Omron CX-Programmer project NewProject (CX-Programmer 9.73)

# PLC FINAL: CS1G CPU42

## Global symbols (name address type ; comment)
C0001 BOOL  ; Reset
C0005 BOOL  ; Brojac ponavljaja
T0001 BOOL  ; Zeleno iskljuceno pesacima
T0002 BOOL  ; Crveno iskljuceno pesacima
T0003 BOOL  ; Zuto iskljuceno kolima
T0004 BOOL  ; Zeleno iskljuceno kolima
T0005 BOOL  ; Brojac

## Program NewProgram1 (cyclic task 0)
Local symbols
Crveno_Pesaci 2961.02 BOOL  ; Pesaci crveno
Crveno_Voz 2961.00 BOOL  ; Lamplica za voz
Crveno_Vozila 2961.01 BOOL  ; Kola Crveno
Flag 200.00 BOOL  ; Voz nije tu
Kraj 2961.06 BOOL  ; Resetuj sistem
Reset 2960.01 BOOL  ; Za startovanje
SV 2960.00 BOOL  ; Voz dolazi
Zeleno_Pesaci 2961.03 BOOL  ; Pesaci zeleno
Zeleno_Vozila 2961.05 BOOL  ; Kola zeleno
Zuto_Vozila 2961.04 BOOL  ; Kola zuto

### Section Section1

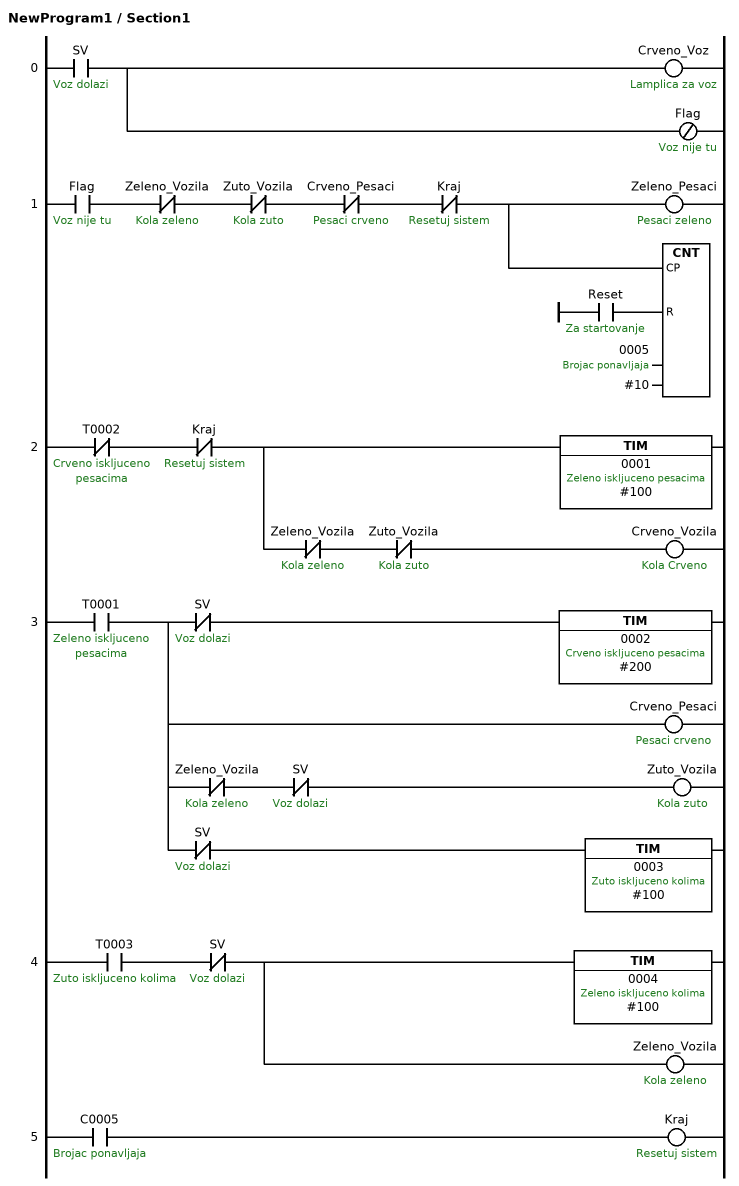
; rung 0
LD SV  ; Voz dolazi
OUT Crveno_Voz  ; Lamplica za voz
OUTNOT Flag  ; Voz nije tu
; rung 1
LD Flag  ; Voz nije tu
ANDNOT Zeleno_Vozila  ; Kola zeleno
ANDNOT Zuto_Vozila  ; Kola zuto
ANDNOT Crveno_Pesaci  ; Pesaci crveno
ANDNOT Kraj  ; Resetuj sistem
OUT Zeleno_Pesaci  ; Pesaci zeleno
LD Reset  ; Za startovanje
CNT 0005 #10  ; Brojac ponavljaja
; rung 2
LDNOT T0002  ; Crveno iskljuceno pesacima
ANDNOT Kraj  ; Resetuj sistem
TIM 0001 #100  ; Zeleno iskljuceno pesacima
ANDNOT Zeleno_Vozila  ; Kola zeleno
ANDNOT Zuto_Vozila  ; Kola zuto
OUT Crveno_Vozila  ; Kola Crveno
; rung 3
LD T0001  ; Zeleno iskljuceno pesacima
OUT TR0
ANDNOT SV  ; Voz dolazi
TIM 0002 #200  ; Crveno iskljuceno pesacima
LD TR0
OUT Crveno_Pesaci  ; Pesaci crveno
ANDNOT Zeleno_Vozila  ; Kola zeleno
ANDNOT SV  ; Voz dolazi
OUT Zuto_Vozila  ; Kola zuto
LD TR0
ANDNOT SV  ; Voz dolazi
TIM 0003 #100  ; Zuto iskljuceno kolima
; rung 4
LD T0003  ; Zuto iskljuceno kolima
ANDNOT SV  ; Voz dolazi
TIM 0004 #100  ; Zeleno iskljuceno kolima
OUT Zeleno_Vozila  ; Kola zeleno
; rung 5
LD C0005  ; Brojac ponavljaja
OUT Kraj  ; Resetuj sistem

### Section END
; rung 0
END(001)